TYPE ST_TcpCodeReaderOutImm :
STRUCT
    LinkState    : E_ByteChannelState;
    LastResponse : STRING(255);
END_STRUCT
END_TYPE

(* stored: Version 1.1.0.1, ProductVersion 3.1.4024.12
   DUT ST_TcpCodeReaderOutImm: Id {379fb691-3f82-416e-8cd7-d68d58278fb6} *)
